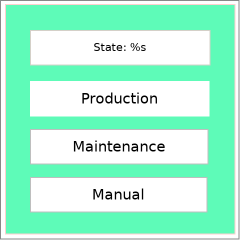
VISUALIZATION V_ChangeMode  // 240x240
VAR_IN_OUT
	HMI : ST_PackMLBaseModule_HMI;
END_VAR
    RoundedRectangle (5,4 230x230)
    Textfield (30,30 180x35), "State: %s", text variable: HMI.Status.State
    RoundedRectangle (30,81 179x35), "Production", colour toggle: HMI.Status.Mode = E_PMLUnitMode.ePMLUnitMode_Production
        OnMouseClick: execute { HMI.Command.Mode := E_PMLUnitMode.ePMLUnitMode_Production; }
    RoundedRectangle (30,129 178x35), "Maintenance", colour toggle: HMI.Status.Mode = E_PMLUnitMode.ePMLUnitMode_Maintenance
        OnMouseClick: execute { HMI.Command.Mode := E_PMLUnitMode.ePMLUnitMode_Maintenance; }
    RoundedRectangle (30,177 177x35), "Manual", colour toggle: HMI.Status.Mode = E_PMLUnitMode.ePMLUnitMode_Manual
        OnMouseClick: execute { HMI.Command.Mode := E_PMLUnitMode.ePMLUnitMode_Manual; }
END_VISUALIZATION

(* stored: Version 1.1.0.1, ProductVersion 3.1.4024.15
   Visu V_ChangeMode: Id {a579ab76-3dfa-0e50-1e72-1a62fe47c520} *)
